	X =  -173.041  mm,	Y =   306.461  mm,	Z =     0.000  mm,
	W =  -167.372 deg,	P =    -0.003 deg,	R =  -135.227 deg
};
P[1118]{
   GP1:
	UF : 7, UT : 3,	CONFIG : 'F U T, 0, 0, 0',
	X =  -173.041  mm,	Y =   306.461  mm,	Z =     0.000  mm,
	W =  -167.372 deg,	P =    -0.003 deg,	R =  -135.227 deg
};
P[1119]{
   GP1:
	UF : 7, UT : 3,	CONFIG : 'F U T, 0, 0, 0',
	X =  -190.720  mm,	Y =   295.790  mm,	Z =     0.003  mm,
	W =  -167.372 deg,	P =    -0.002 deg,	R =  -132.163 deg
};
P[1120]{
   GP1:
	UF : 7, UT : 3,	CONFIG : 'F U T, 0, 0, 0',
	X =  -206.490  mm,	Y =   284.994  mm,	Z =     0.009  mm,
	W =  -167.373 deg,	P =    -0.002 deg,	R =  -128.960 deg
};
P[1121]{
   GP1:
	UF : 7, UT : 3,	CONFIG : 'F U T, 0, 0, 0',
	X =  -222.160  mm,	Y =   272.963  mm,	Z =     0.016  mm,
	W =  -167.373 deg,	P =    -0.001 deg,	R =  -125.844 deg
};
P[1122]{
   GP1:
	UF : 7, UT : 3,	CONFIG : 'F U T, 0, 0, 0',
	X =  -236.698  mm,	Y =   260.451  mm,	Z =     0.021  mm,
	W =  -167.374 deg,	P =     0.000 deg,	R =  -122.644 deg
};
P[1123]{
   GP1:
	UF : 7, UT : 3,	CONFIG : 'F U T, 0, 0, 0',
	X =  -249.147  mm,	Y =   248.563  mm,	Z =     0.016  mm,
	W =  -167.414 deg,	P =     0.050 deg,	R =  -119.969 deg
};
P[1124]{
   GP1:
	UF : 7, UT : 3,	CONFIG : 'F U T, 0, 0, 0',
	X =  -260.264  mm,	Y =   236.898  mm,	Z =     0.000  mm,
	W =  -167.447 deg,	P =     0.100 deg,	R =  -117.131 deg
};
P[1125]{
   GP1:
	UF : 7, UT : 3,	CONFIG : 'F U T, 0, 0, 0',
	X =  -260.264  mm,	Y =   236.898  mm,	Z =     0.000  mm,
	W =  -167.447 deg,	P =     0.100 deg,	R =  -117.131 deg
};
P[1126]{
   GP1:
	UF : 7, UT : 3,	CONFIG : 'F U T, 0, 0, 0',
	X =  -260.264  mm,	Y =   236.898  mm,	Z =     0.000  mm,
	W =  -167.447 deg,	P =     0.100 deg,	R =  -117.131 deg
};
P[1127]{
   GP1:
	UF : 7, UT : 3,	CONFIG : 'F U T, 0, 0, 0',
	X =  -260.264  mm,	Y =   236.898  mm,	Z =     0.000  mm,
	W =  -167.447 deg,	P =     0.100 deg,	R =  -117.131 deg
};
P[1128]{
   GP1:
	UF : 7, UT : 3,	CONFIG : 'F U T, 0, 0, 0',
	X =  -288.873  mm,	Y =   201.022  mm,	Z =     0.000  mm,
	W =  -167.893 deg,	P =    -0.197 deg,	R =  -110.313 deg
};
P[1129]{
   GP1:
	UF : 7, UT : 3,	CONFIG : 'F U T, 0, 0, 0',
	X =  -288.873  mm,	Y =   201.022  mm,	Z =     0.000  mm,
	W =  -167.893 deg,	P =    -0.197 deg,	R =  -110.313 deg
};
P[1130]{
   GP1:
	UF : 7, UT : 3,	CONFIG : 'F U T, 0, 0, 0',
	X =  -288.873  mm,	Y =   201.022  mm,	Z =     0.000  mm,
	W =  -167.893 deg,	P =    -0.197 deg,	R =  -110.313 deg
};
P[1131]{
   GP1:
	UF : 7, UT : 3,	CONFIG : 'F U T, 0, 0, 0',
	X =  -288.873  mm,	Y =   201.022  mm,	Z =     0.000  mm,
	W =  -167.893 deg,	P =    -0.197 deg,	R =  -110.313 deg
};
P[1132]{
   GP1:
	UF : 7, UT : 3,	CONFIG : 'F U T, 0, 0, 0',
	X =  -297.890  mm,	Y =   187.407  mm,	Z =     0.208  mm,
	W =  -168.125 deg,	P =    -1.096 deg,	R =  -107.109 deg
};
P[1133]{
   GP1:
	UF : 7, UT : 3,	CONFIG : 'F U T, 0, 0, 0',
	X =  -301.777  mm,	Y =   181.079  mm,	Z =     0.410  mm,
	W =  -168.208 deg,	P =    -1.678 deg,	R =  -106.017 deg
};
P[1134]{
   GP1:
	UF : 7, UT : 3,	CONFIG : 'F U T, 0, 0, 0',
	X =  -306.225  mm,	Y =   173.464  mm,	Z =     0.720  mm,
	W =  -168.359 deg,	P =    -1.852 deg,	R =  -104.630 deg
};
P[1135]{
   GP1:
	UF : 7, UT : 3,	CONFIG : 'F U T, 0, 0, 0',
	X =  -310.479  mm,	Y =   165.757  mm,	Z =     1.000  mm,
	W =  -168.472 deg,	P =    -1.237 deg,	R =  -103.508 deg
};
P[1136]{
   GP1:
	UF : 7, UT : 3,	CONFIG : 'F U T, 0, 0, 0',
	X =  -310.479  mm,	Y =   165.757  mm,	Z =     1.000  mm,
	W =  -168.472 deg,	P =    -1.237 deg,	R =  -103.508 deg
};
P[1137]{
   GP1:
	UF : 7, UT : 3,	CONFIG : 'F U T, 0, 0, 0',
	X =  -310.479  mm,	Y =   165.757  mm,	Z =     1.000  mm,
	W =  -168.472 deg,	P =    -1.237 deg,	R =  -103.508 deg
};
P[1138]{
   GP1:
	UF : 7, UT : 3,	CONFIG : 'F U T, 0, 0, 0',
	X =  -310.479  mm,	Y =   165.757  mm,	Z =     1.000  mm,
	W =  -168.472 deg,	P =    -1.237 deg,	R =  -103.508 deg
};
P[1139]{
   GP1:
	UF : 7, UT : 3,	CONFIG : 'F U T, 0, 0, 0',
	X =  -323.165  mm,	Y =   139.394  mm,	Z =     1.000  mm,
	W =  -167.595 deg,	P =     1.008 deg,	R =   -98.966 deg
};
P[1140]{
   GP1:
	UF : 7, UT : 3,	CONFIG : 'F U T, 0, 0, 0',
	X =  -323.165  mm,	Y =   139.394  mm,	Z =     1.000  mm,
	W =  -167.595 deg,	P =     1.008 deg,	R =   -98.966 deg
};
P[1141]{
   GP1:
	UF : 7, UT : 3,	CONFIG : 'F U T, 0, 0, 0',
	X =  -323.165  mm,	Y =   139.394  mm,	Z =     1.000  mm,
	W =  -167.595 deg,	P =     1.008 deg,	R =   -98.966 deg
};
P[1142]{
   GP1:
	UF : 7, UT : 3,	CONFIG : 'F U T, 0, 0, 0',
	X =  -323.165  mm,	Y =   139.394  mm,	Z =     1.000  mm,
	W =  -167.595 deg,	P =     1.008 deg,	R =   -98.966 deg
};
P[1143]{
   GP1:
	UF : 7, UT : 3,	CONFIG : 'F U T, 0, 0, 0',
	X =  -328.405  mm,	Y =   126.540  mm,	Z =     0.631  mm,
	W =  -167.514 deg,	P =     2.212 deg,	R =   -95.957 deg
};
P[1144]{
   GP1:
	UF : 7, UT : 3,	CONFIG : 'F U T, 0, 0, 0',
	X =  -330.738  mm,	Y =   120.311  mm,	Z =     0.385  mm,
	W =  -167.607 deg,	P =     2.141 deg,	R =   -94.815 deg
};
P[1145]{
   GP1:
	UF : 7, UT : 3,	CONFIG : 'F U T, 0, 0, 0',
	X =  -335.864  mm,	Y =   105.155  mm,	Z =     0.029  mm,
	W =  -167.677 deg,	P =     0.615 deg,	R =   -92.305 deg
};
P[1146]{
   GP1:
	UF : 7, UT : 3,	CONFIG : 'F U T, 0, 0, 0',
	X =  -337.294  mm,	Y =   100.499  mm,	Z =     0.000  mm,
	W =  -167.622 deg,	P =     0.306 deg,	R =   -92.059 deg
};
P[1147]{
   GP1:
	UF : 7, UT : 3,	CONFIG : 'F U T, 0, 0, 0',
	X =  -337.294  mm,	Y =   100.499  mm,	Z =     0.000  mm,
	W =  -167.622 deg,	P =     0.306 deg,	R =   -92.059 deg
};
P[1148]{
   GP1:
	UF : 7, UT : 3,	CONFIG : 'F U T, 0, 0, 0',
	X =  -337.294  mm,	Y =   100.499  mm,	Z =     0.000  mm,
	W =  -167.622 deg,	P =     0.306 deg,	R =   -92.059 deg
};
P[1149]{
   GP1:
	UF : 7, UT : 3,	CONFIG : 'F U T, 0, 0, 0',
	X =  -337.294  mm,	Y =   100.499  mm,	Z =     0.000  mm,
	W =  -167.622 deg,	P =     0.306 deg,	R =   -92.059 deg
};
P[1150]{
   GP1:
	UF : 7, UT : 3,	CONFIG : 'F U T, 0, 1, 0',
	X =  -347.491  mm,	Y =    55.790  mm,	Z =     0.000  mm,
	W =  -167.390 deg,	P =    -0.010 deg,	R =   -84.124 deg
};
P[1151]{
   GP1:
	UF : 7, UT : 3,	CONFIG : 'F U T, 0, 1, 0',
	X =  -347.491  mm,	Y =    55.790  mm,	Z =     0.000  mm,
	W =  -167.390 deg,	P =    -0.010 deg,	R =   -84.124 deg
};
P[1152]{
   GP1:
	UF : 7, UT : 3,	CONFIG : 'F U T, 0, 1, 0',
	X =  -347.491  mm,	Y =    55.790  mm,	Z =     0.000  mm,
	W =  -167.390 deg,	P =    -0.010 deg,	R =   -84.124 deg
};
P[1153]{
   GP1:
	UF : 7, UT : 3,	CONFIG : 'F U T, 0, 1, 0',
	X =  -347.491  mm,	Y =    55.790  mm,	Z =     0.000  mm,
	W =  -167.390 deg,	P =    -0.010 deg,	R =   -84.124 deg
};
P[1154]{
   GP1:
	UF : 7, UT : 3,	CONFIG : 'F U T, 0, 1, 0',
	X =  -349.820  mm,	Y =    38.586  mm,	Z =     0.003  mm,
	W =  -167.382 deg,	P =    -0.003 deg,	R =   -81.231 deg
};
P[1155]{
   GP1:
	UF : 7, UT : 3,	CONFIG : 'F U T, 0, 1, 0',
	X =  -351.303  mm,	Y =    21.167  mm,	Z =     0.003  mm,
	W =  -167.373 deg,	P =     0.003 deg,	R =   -78.345 deg
};
P[1156]{
   GP1:
	UF : 7, UT : 3,	CONFIG : 'F U T, 0, 1, 0',
	X =  -351.955  mm,	Y =     0.000  mm,	Z =     0.000  mm,
	W =  -167.361 deg,	P =     0.009 deg,	R =   -75.581 deg
};
P[1157]{
   GP1:
	UF : 7, UT : 3,	CONFIG : 'F U T, 0, 1, 0',
	X =  -351.955  mm,	Y =     0.000  mm,	Z =     0.000  mm,
	W =  -167.361 deg,	P =     0.009 deg,	R =   -75.581 deg
};
P[1158]{
   GP1:
	UF : 7, UT : 3,	CONFIG : 'F U T, 0, 1, 0',
	X =  -351.955  mm,	Y =     0.000  mm,	Z =     0.000  mm,
	W =  -167.361 deg,	P =     0.009 deg,	R =   -75.581 deg
};
P[1159]{
   GP1:
	UF : 7, UT : 3,	CONFIG : 'F U T, 0, 1, 0',
	X =  -351.955  mm,	Y =     0.000  mm,	Z =     0.000  mm,
	W =  -167.361 deg,	P =     0.009 deg,	R =   -75.581 deg
};
P[1160]{
   GP1:
	UF : 7, UT : 3,	CONFIG : 'F U T, 0, 1, 0',
	X =  -348.821  mm,	Y =     0.000  mm,	Z =     0.000  mm,
	W =  -167.361 deg,	P =     0.009 deg,	R =   -75.580 deg
};
P[1161]{
   GP1:
	UF : 7, UT : 3,	CONFIG : 'F U T, 0, 1, 0',
	X =  -348.821  mm,	Y =     0.000  mm,	Z =     0.000  mm,
	W =  -167.361 deg,	P =     0.009 deg,	R =   -75.580 deg
};
P[1162]{
   GP1:
	UF : 7, UT : 3,	CONFIG : 'F U T, 0, 1, 0',
	X =  -348.821  mm,	Y =     0.000  mm,	Z =     0.000  mm,
	W =  -167.361 deg,	P =     0.009 deg,	R =   -75.580 deg
};
P[1163]{
   GP1:
	UF : 7, UT : 3,	CONFIG : 'F U T, 0, 1, 0',
	X =  -348.821  mm,	Y =     0.000  mm,	Z =     0.000  mm,
	W =  -167.361 deg,	P =     0.009 deg,	R =   -75.580 deg
};
P[1164]{
   GP1:
	UF : 7, UT : 3,	CONFIG : 'F U T, 0, 1, 0',
	X =  -347.719  mm,	Y =    27.446  mm,	Z =     0.003  mm,
	W =  -167.374 deg,	P =    -0.001 deg,	R =   -79.422 deg
};
P[1165]{
   GP1:
	UF : 7, UT : 3,	CONFIG : 'F U T, 0, 1, 0',
	X =  -344.991  mm,	Y =    51.425  mm,	Z =     0.000  mm,
	W =  -167.384 deg,	P =    -0.011 deg,	R =   -83.308 deg
};
P[1166]{
   GP1:
	UF : 7, UT : 3,	CONFIG : 'F U T, 0, 1, 0',
	X =  -344.991  mm,	Y =    51.425  mm,	Z =     0.000  mm,
	W =  -167.384 deg,	P =    -0.011 deg,	R =   -83.308 deg
};
P[1167]{
   GP1:
	UF : 7, UT : 3,	CONFIG : 'F U T, 0, 1, 0',
	X =  -344.991  mm,	Y =    51.425  mm,	Z =     0.000  mm,
	W =  -167.384 deg,	P =    -0.011 deg,	R =   -83.308 deg
};
P[1168]{
   GP1:
	UF : 7, UT : 3,	CONFIG : 'F U T, 0, 1, 0',
	X =  -344.991  mm,	Y =    51.425  mm,	Z =     0.000  mm,
	W =  -167.384 deg,	P =    -0.011 deg,	R =   -83.308 deg
};
P[1169]{
   GP1:
	UF : 7, UT : 3,	CONFIG : 'F U T, 0, 0, 0',
	X =  -333.135  mm,	Y =   103.355  mm,	Z =     0.000  mm,
	W =  -167.638 deg,	P =     0.437 deg,	R =   -91.561 deg
};
P[1170]{
   GP1:
	UF : 7, UT : 3,	CONFIG : 'F U T, 0, 0, 0',
	X =  -333.135  mm,	Y =   103.355  mm,	Z =     0.000  mm,
	W =  -167.638 deg,	P =     0.437 deg,	R =   -91.561 deg
};
P[1171]{
   GP1:
	UF : 7, UT : 3,	CONFIG : 'F U T, 0, 0, 0',
	X =  -333.135  mm,	Y =   103.355  mm,	Z =     0.000  mm,
	W =  -167.638 deg,	P =     0.437 deg,	R =   -91.561 deg
};
P[1172]{
   GP1:
	UF : 7, UT : 3,	CONFIG : 'F U T, 0, 0, 0',
	X =  -333.135  mm,	Y =   103.355  mm,	Z =     0.000  mm,
	W =  -167.638 deg,	P =     0.437 deg,	R =   -91.561 deg
};
P[1173]{
   GP1:
	UF : 7, UT : 3,	CONFIG : 'F U T, 0, 0, 0',
	X =  -328.255  mm,	Y =   117.948  mm,	Z =     0.291  mm,
	W =  -167.684 deg,	P =     2.047 deg,	R =   -94.688 deg
};
P[1174]{
   GP1:
	UF : 7, UT : 3,	CONFIG : 'F U T, 0, 0, 0',
	X =  -325.878  mm,	Y =   124.367  mm,	Z =     0.545  mm,
	W =  -167.629 deg,	P =     2.346 deg,	R =   -95.800 deg
};
P[1175]{
   GP1:
	UF : 7, UT : 3,	CONFIG : 'F U T, 0, 0, 0',
	X =  -324.799  mm,	Y =   127.193  mm,	Z =     0.659  mm,
	W =  -167.621 deg,	P =     2.234 deg,	R =   -96.230 deg
};
P[1176]{
   GP1:
	UF : 7, UT : 3,	CONFIG : 'F U T, 0, 0, 0',
	X =  -319.450  mm,	Y =   140.081  mm,	Z =     1.000  mm,
	W =  -167.790 deg,	P =     0.910 deg,	R =   -98.471 deg
};
P[1177]{
   GP1:
	UF : 7, UT : 3,	CONFIG : 'F U T, 0, 0, 0',
	X =  -319.450  mm,	Y =   140.081  mm,	Z =     1.000  mm,
	W =  -167.790 deg,	P =     0.910 deg,	R =   -98.471 deg
};
P[1178]{
   GP1:
	UF : 7, UT : 3,	CONFIG : 'F U T, 0, 0, 0',
	X =  -319.450  mm,	Y =   140.081  mm,	Z =     1.000  mm,
	W =  -167.790 deg,	P =     0.910 deg,	R =   -98.471 deg
};
P[1179]{
   GP1:
	UF : 7, UT : 3,	CONFIG : 'F U T, 0, 0, 0',
	X =  -319.450  mm,	Y =   140.081  mm,	Z =     1.000  mm,
	W =  -167.790 deg,	P =     0.910 deg,	R =   -98.471 deg
};
P[1180]{
   GP1:
	UF : 7, UT : 3,	CONFIG : 'F U T, 0, 0, 0',
	X =  -308.698  mm,	Y =   162.429  mm,	Z =     1.000  mm,
	W =  -168.619 deg,	P =    -0.871 deg,	R =  -102.937 deg
};
P[1181]{
   GP1:
	UF : 7, UT : 3,	CONFIG : 'F U T, 0, 0, 0',
	X =  -308.698  mm,	Y =   162.429  mm,	Z =     1.000  mm,
	W =  -168.619 deg,	P =    -0.871 deg,	R =  -102.937 deg
};
P[1182]{
   GP1:
	UF : 7, UT : 3,	CONFIG : 'F U T, 0, 0, 0',
	X =  -308.698  mm,	Y =   162.429  mm,	Z =     1.000  mm,
	W =  -168.619 deg,	P =    -0.871 deg,	R =  -102.937 deg
};
P[1183]{
   GP1:
	UF : 7, UT : 3,	CONFIG : 'F U T, 0, 0, 0',
	X =  -308.698  mm,	Y =   162.429  mm,	Z =     1.000  mm,
	W =  -168.619 deg,	P =    -0.871 deg,	R =  -102.937 deg
};
P[1184]{
   GP1:
	UF : 7, UT : 3,	CONFIG : 'F U T, 0, 0, 0',
	X =  -304.278  mm,	Y =   170.562  mm,	Z =     0.741  mm,
	W =  -168.545 deg,	P =    -1.673 deg,	R =  -104.288 deg
};
P[1185]{
   GP1:
	UF : 7, UT : 3,	CONFIG : 'F U T, 0, 0, 0',
	X =  -299.991  mm,	Y =   177.979  mm,	Z =     0.443  mm,
	W =  -168.362 deg,	P =    -1.726 deg,	R =  -105.695 deg
};
P[1186]{
   GP1:
	UF : 7, UT : 3,	CONFIG : 'F U T, 0, 0, 0',
	X =  -288.517  mm,	Y =   196.042  mm,	Z =     0.000  mm,
	W =  -167.992 deg,	P =    -0.314 deg,	R =  -108.539 deg
};
P[1187]{
   GP1:
	UF : 7, UT : 3,	CONFIG : 'F U T, 0, 0, 0',
	X =  -288.517  mm,	Y =   196.042  mm,	Z =     0.000  mm,
	W =  -167.992 deg,	P =    -0.314 deg,	R =  -108.539 deg
};
P[1188]{
   GP1:
	UF : 7, UT : 3,	CONFIG : 'F U T, 0, 0, 0',
	X =  -288.517  mm,	Y =   196.042  mm,	Z =     0.000  mm,
	W =  -167.992 deg,	P =    -0.314 deg,	R =  -108.539 deg
};
P[1189]{
   GP1:
	UF : 7, UT : 3,	CONFIG : 'F U T, 0, 0, 0',
	X =  -288.517  mm,	Y =   196.042  mm,	Z =     0.000  mm,
	W =  -167.992 deg,	P =    -0.314 deg,	R =  -108.539 deg
};
P[1190]{
   GP1:
	UF : 7, UT : 3,	CONFIG : 'F U T, 0, 0, 0',
	X =  -255.318  mm,	Y =   237.661  mm,	Z =     0.000  mm,
	W =  -167.431 deg,	P =     0.104 deg,	R =  -118.108 deg
};
P[1191]{
   GP1:
	UF : 7, UT : 3,	CONFIG : 'F U T, 0, 0, 0',
	X =  -255.318  mm,	Y =   237.661  mm,	Z =     0.000  mm,
	W =  -167.431 deg,	P =     0.104 deg,	R =  -118.108 deg
};
P[1192]{
   GP1:
	UF : 7, UT : 3,	CONFIG : 'F U T, 0, 0, 0',
	X =  -255.318  mm,	Y =   237.661  mm,	Z =     0.000  mm,
	W =  -167.431 deg,	P =     0.104 deg,	R =  -118.108 deg
};
P[1193]{
   GP1:
	UF : 7, UT : 3,	CONFIG : 'F U T, 0, 0, 0',
	X =  -255.318  mm,	Y =   237.661  mm,	Z =     0.000  mm,
	W =  -167.431 deg,	P =     0.104 deg,	R =  -118.108 deg
};
P[1194]{
   GP1:
	UF : 7, UT : 3,	CONFIG : 'F U T, 0, 0, 0',
	X =  -244.166  mm,	Y =   249.102  mm,	Z =     0.017  mm,
	W =  -167.403 deg,	P =     0.049 deg,	R =  -120.505 deg
};
P[1195]{
   GP1:
	UF : 7, UT : 3,	CONFIG : 'F U T, 0, 0, 0',
	X =  -232.964  mm,	Y =   259.606  mm,	Z =     0.020  mm,
	W =  -167.373 deg,	P =    -0.001 deg,	R =  -123.022 deg
};
P[1196]{
   GP1:
	UF : 7, UT : 3,	CONFIG : 'F U T, 0, 0, 0',
	X =  -219.177  mm,	Y =   271.343  mm,	Z =     0.016  mm,
	W =  -167.373 deg,	P =    -0.002 deg,	R =  -126.041 deg
};
P[1197]{
   GP1:
	UF : 7, UT : 3,	CONFIG : 'F U T, 0, 0, 0',
	X =  -204.531  mm,	Y =   282.545  mm,	Z =     0.009  mm,
	W =  -167.373 deg,	P =    -0.003 deg,	R =  -129.005 deg
};
P[1198]{
   GP1:
	UF : 7, UT : 3,	CONFIG : 'F U T, 0, 0, 0',
	X =  -189.632  mm,	Y =   292.762  mm,	Z =     0.003  mm,
	W =  -167.373 deg,	P =    -0.004 deg,	R =  -132.024 deg
};
P[1199]{
   GP1:
	UF : 7, UT : 3,	CONFIG : 'F U T, 0, 0, 0',
	X =  -174.892  mm,	Y =   301.790  mm,	Z =     0.000  mm,
	W =  -167.372 deg,	P =    -0.005 deg,	R =  -135.243 deg
};
P[1200]{
   GP1:
	UF : 7, UT : 3,	CONFIG : 'F U T, 0, 0, 0',
	X =  -174.892  mm,	Y =   301.790  mm,	Z =     0.000  mm,
	W =  -167.372 deg,	P =    -0.005 deg,	R =  -135.243 deg
};
P[1201]{
   GP1:
	UF : 7, UT : 3,	CONFIG : 'F U T, 0, 0, 0',
	X =  -174.892  mm,	Y =   301.790  mm,	Z =     0.000  mm,
	W =  -167.372 deg,	P =    -0.005 deg,	R =  -135.243 deg
};
P[1202]{
   GP1:
	UF : 7, UT : 3,	CONFIG : 'F U T, 0, 0, 0',
	X =  -174.892  mm,	Y =   301.790  mm,	Z =     0.000  mm,
	W =  -167.372 deg,	P =    -0.005 deg,	R =  -135.243 deg
};
P[1203]{
   GP1:
	UF : 7, UT : 3,	CONFIG : 'F U T, 0, 0, 0',
	X =  -126.912  mm,	Y =   324.901  mm,	Z =     0.000  mm,
	W =  -167.365 deg,	P =     0.002 deg,	R =  -144.020 deg
};
P[1204]{
   GP1:
	UF : 7, UT : 3,	CONFIG : 'F U T, 0, 0, 0',
	X =  -126.912  mm,	Y =   324.901  mm,	Z =     0.000  mm,
	W =  -167.365 deg,	P =     0.002 deg,	R =  -144.020 deg
};
P[1205]{
   GP1:
	UF : 7, UT : 3,	CONFIG : 'F U T, 0, 0, 0',
	X =  -126.912  mm,	Y =   324.901  mm,	Z =     0.000  mm,
	W =  -167.365 deg,	P =     0.002 deg,	R =  -144.020 deg
};
P[1206]{
   GP1:
	UF : 7, UT : 3,	CONFIG : 'F U T, 0, 0, 0',
	X =  -126.912  mm,	Y =   324.901  mm,	Z =     0.000  mm,
	W =  -167.365 deg,	P =     0.002 deg,	R =  -144.020 deg
};
P[1207]{
   GP1:
	UF : 7, UT : 3,	CONFIG : 'F U T, 0, 0, 0',
	X =  -106.083  mm,	Y =   332.287  mm,	Z =     0.000  mm,
	W =  -167.364 deg,	P =     0.001 deg,	R =  -147.250 deg
};
P[1208]{
   GP1:
	UF : 7, UT : 3,	CONFIG : 'F U T, 0, 0, 0',
	X =   -88.319  mm,	Y =   337.433  mm,	Z =     0.000  mm,
	W =  -167.363 deg,	P =     0.000 deg,	R =  -150.913 deg
};
P[1209]{
   GP1:
	UF : 7, UT : 3,	CONFIG : 'F U T, 0, 0, 0',
	X =   -88.319  mm,	Y =   337.433  mm,	Z =     0.000  mm,
	W =  -167.363 deg,	P =     0.000 deg,	R =  -150.913 deg
};
P[1210]{
   GP1:
	UF : 7, UT : 3,	CONFIG : 'F U T, 0, 0, 0',
	X =   -88.319  mm,	Y =   337.433  mm,	Z =     0.000  mm,
	W =  -167.363 deg,	P =     0.000 deg,	R =  -150.913 deg
};
P[1211]{
   GP1:
	UF : 7, UT : 3,	CONFIG : 'F U T, 0, 0, 0',
	X =   -88.319  mm,	Y =   337.433  mm,	Z =     0.000  mm,
	W =  -167.363 deg,	P =     0.000 deg,	R =  -150.913 deg
};
P[1212]{
   GP1:
	UF : 7, UT : 3,	CONFIG : 'F U T, 0, 0, 0',
	X =   -66.816  mm,	Y =   342.344  mm,	Z =     0.000  mm,
	W =  -167.363 deg,	P =     0.000 deg,	R =  -154.099 deg
};
P[1213]{
   GP1:
	UF : 7, UT : 3,	CONFIG : 'F U T, 0, 0, 0',
	X =   -66.816  mm,	Y =   342.344  mm,	Z =     0.000  mm,
	W =  -167.363 deg,	P =     0.000 deg,	R =  -154.099 deg
};
P[1214]{
   GP1:
	UF : 7, UT : 3,	CONFIG : 'F U T, 0, 0, 0',
	X =   -66.816  mm,	Y =   342.344  mm,	Z =     0.000  mm,
	W =  -167.363 deg,	P =     0.000 deg,	R =  -154.099 deg
};
P[1215]{
   GP1:
	UF : 7, UT : 3,	CONFIG : 'F U T, 0, 0, 0',
	X =   -66.816  mm,	Y =   342.344  mm,	Z =     0.000  mm,
	W =  -167.363 deg,	P =     0.000 deg,	R =  -154.099 deg
};
P[1216]{
   GP1:
	UF : 7, UT : 3,	CONFIG : 'F U T, 0, 0, 0',
	X =   -46.005  mm,	Y =   345.765  mm,	Z =     0.000  mm,
	W =  -167.363 deg,	P =     0.000 deg,	R =  -157.374 deg
};
P[1217]{
   GP1:
	UF : 7, UT : 3,	CONFIG : 'F U T, 0, 0, 0',
	X =   -26.635  mm,	Y =   347.781  mm,	Z =     0.000  mm,
	W =  -167.364 deg,	P =     0.000 deg,	R =  -160.858 deg
};
P[1218]{
   GP1:
	UF : 7, UT : 3,	CONFIG : 'F U T, 0, 0, 0',
	X =   -26.635  mm,	Y =   347.781  mm,	Z =     0.000  mm,
	W =  -167.364 deg,	P =     0.000 deg,	R =  -160.858 deg
};
P[1219]{
   GP1:
	UF : 7, UT : 3,	CONFIG : 'F U T, 0, 0, 0',
	X =   -26.635  mm,	Y =   347.781  mm,	Z =     0.000  mm,
	W =  -167.364 deg,	P =     0.000 deg,	R =  -160.858 deg
};
P[1220]{
   GP1:
	UF : 7, UT : 3,	CONFIG : 'F U T, 0, 0, 0',
	X =   -26.635  mm,	Y =   347.781  mm,	Z =     0.000  mm,
	W =  -167.364 deg,	P =     0.000 deg,	R =  -160.858 deg
};
P[1221]{
   GP1:
	UF : 7, UT : 3,	CONFIG : 'F U T, 0, 0, 0',
	X =    26.635  mm,	Y =   347.781  mm,	Z =     0.000  mm,
	W =  -167.363 deg,	P =     0.000 deg,	R =  -169.046 deg
};
P[1222]{
   GP1:
	UF : 7, UT : 3,	CONFIG : 'F U T, 0, 0, 0',
	X =    26.635  mm,	Y =   347.781  mm,	Z =     0.000  mm,
	W =  -167.363 deg,	P =     0.000 deg,	R =  -169.046 deg
};
P[1223]{
   GP1:
	UF : 7, UT : 3,	CONFIG : 'F U T, 0, 0, 0',
	X =    26.635  mm,	Y =   347.781  mm,	Z =     0.000  mm,
	W =  -167.363 deg,	P =     0.000 deg,	R =  -169.046 deg
};
P[1224]{
   GP1:
	UF : 7, UT : 3,	CONFIG : 'F U T, 0, 0, 0',
	X =    26.635  mm,	Y =   347.781  mm,	Z =     0.000  mm,
	W =  -167.363 deg,	P =     0.000 deg,	R =  -169.046 deg
};
P[1225]{
   GP1:
	UF : 7, UT : 3,	CONFIG : 'F U T, 0, 0, 0',
	X =    45.934  mm,	Y =   345.776  mm,	Z =     0.000  mm,
	W =  -167.363 deg,	P =     0.000 deg,	R =  -172.500 deg
};
P[1226]{
   GP1:
	UF : 7, UT : 3,	CONFIG : 'F U T, 0, 0, 0',
	X =    66.816  mm,	Y =   342.344  mm,	Z =     0.000  mm,
	W =  -167.363 deg,	P =     0.000 deg,	R =  -175.771 deg
};
P[1227]{
   GP1:
	UF : 7, UT : 3,	CONFIG : 'F U T, 0, 0, 0',
	X =    66.816  mm,	Y =   342.344  mm,	Z =     0.000  mm,
	W =  -167.363 deg,	P =     0.000 deg,	R =  -175.771 deg
};
P[1228]{
   GP1:
	UF : 7, UT : 3,	CONFIG : 'F U T, 0, 0, 0',
	X =    66.816  mm,	Y =   342.344  mm,	Z =     0.000  mm,
	W =  -167.363 deg,	P =     0.000 deg,	R =  -175.771 deg
};
P[1229]{
   GP1:
	UF : 7, UT : 3,	CONFIG : 'F U T, 0, 0, 0',
	X =    66.816  mm,	Y =   342.344  mm,	Z =     0.000  mm,
	W =  -167.363 deg,	P =     0.000 deg,	R =  -175.771 deg
};
P[1230]{
   GP1:
	UF : 7, UT : 3,	CONFIG : 'F U T, 0, 0, 0',
	X =    88.319  mm,	Y =   337.433  mm,	Z =     0.000  mm,
	W =  -167.363 deg,	P =     0.000 deg,	R =  -179.012 deg
};
P[1231]{
   GP1:
	UF : 7, UT : 3,	CONFIG : 'F U T, 0, 0, 0',
	X =    88.319  mm,	Y =   337.433  mm,	Z =     0.000  mm,
	W =  -167.363 deg,	P =     0.000 deg,	R =  -179.012 deg
};
P[1232]{
   GP1:
	UF : 7, UT : 3,	CONFIG : 'F U T, 0, 0, 0',
	X =    88.319  mm,	Y =   337.433  mm,	Z =     0.000  mm,
	W =  -167.363 deg,	P =     0.000 deg,	R =  -179.012 deg
};
P[1233]{
   GP1:
	UF : 7, UT : 3,	CONFIG : 'F U T, 0, 0, 0',
	X =    88.319  mm,	Y =   337.433  mm,	Z =     0.000  mm,
	W =  -167.363 deg,	P =     0.000 deg,	R =  -179.012 deg
};
P[1234]{
   GP1:
	UF : 7, UT : 3,	CONFIG : 'F U T, 0, 0, 0',
	X =   106.083  mm,	Y =   332.287  mm,	Z =     0.000  mm,
	W =  -167.364 deg,	P =     0.000 deg,	R =   177.374 deg
};
P[1235]{
   GP1:
	UF : 7, UT : 3,	CONFIG : 'F U T, 0, 0, 0',
	X =   126.912  mm,	Y =   324.901  mm,	Z =     0.000  mm,
	W =  -167.364 deg,	P =     0.000 deg,	R =   174.134 deg
};
P[1236]{
   GP1:
	UF : 7, UT : 3,	CONFIG : 'F U T, 0, 0, 0',
	X =   126.912  mm,	Y =   324.901  mm,	Z =     0.000  mm,
	W =  -167.364 deg,	P =     0.000 deg,	R =   174.134 deg
};
P[1237]{
   GP1:
	UF : 7, UT : 3,	CONFIG : 'F U T, 0, 0, 0',
	X =   126.912  mm,	Y =   324.901  mm,	Z =     0.000  mm,
	W =  -167.364 deg,	P =     0.000 deg,	R =   174.134 deg
};
P[1238]{
   GP1:
	UF : 7, UT : 3,	CONFIG : 'F U T, 0, 0, 0',
	X =   126.912  mm,	Y =   324.901  mm,	Z =     0.000  mm,
	W =  -167.364 deg,	P =     0.000 deg,	R =   174.134 deg
};
P[1239]{
   GP1:
	UF : 7, UT : 3,	CONFIG : 'F U T, 0, 0, 0',
	X =   174.892  mm,	Y =   301.790  mm,	Z =     0.000  mm,
	W =  -167.364 deg,	P =     0.001 deg,	R =   165.335 deg
};
P[1240]{
   GP1:
	UF : 7, UT : 3,	CONFIG : 'F U T, 0, 0, 0',
	X =   174.892  mm,	Y =   301.790  mm,	Z =     0.000  mm,
	W =  -167.364 deg,	P =     0.001 deg,	R =   165.335 deg
};
P[1241]{
   GP1:
	UF : 7, UT : 3,	CONFIG : 'F U T, 0, 0, 0',
	X =   174.892  mm,	Y =   301.790  mm,	Z =     0.000  mm,
	W =  -167.364 deg,	P =     0.001 deg,	R =   165.335 deg
};
P[1242]{
   GP1:
	UF : 7, UT : 3,	CONFIG : 'F U T, 0, 0, 0',
	X =   174.892  mm,	Y =   301.790  mm,	Z =     0.000  mm,
	W =  -167.364 deg,	P =     0.001 deg,	R =   165.335 deg
};
P[1243]{
   GP1:
	UF : 7, UT : 3,	CONFIG : 'F U T, 0, 0, 0',
	X =   191.564  mm,	Y =   291.498  mm,	Z =     0.000  mm,
	W =  -167.364 deg,	P =     0.000 deg,	R =   161.703 deg
};
P[1244]{
   GP1:
	UF : 7, UT : 3,	CONFIG : 'F U T, 0, 0, 0',
	X =   208.616  mm,	Y =   279.549  mm,	Z =     0.000  mm,
	W =  -167.364 deg,	P =     0.000 deg,	R =   158.339 deg
};
P[1245]{
   GP1:
	UF : 7, UT : 3,	CONFIG : 'F U T, 0, 0, 0',
	X =   224.914  mm,	Y =   266.601  mm,	Z =     0.001  mm,
	W =  -167.364 deg,	P =     0.000 deg,	R =   154.951 deg
};
P[1246]{
   GP1:
	UF : 7, UT : 3,	CONFIG : 'F U T, 0, 0, 0',
	X =   239.976  mm,	Y =   253.131  mm,	Z =     0.000  mm,
	W =  -167.365 deg,	P =     0.000 deg,	R =   151.474 deg
};
P[1247]{
   GP1:
	UF : 7, UT : 3,	CONFIG : 'F U T, 0, 0, 0',
	X =   255.318  mm,	Y =   237.661  mm,	Z =     0.000  mm,
	W =  -167.365 deg,	P =    -0.001 deg,	R =   148.214 deg
};
P[1248]{
   GP1:
	UF : 7, UT : 3,	CONFIG : 'F U T, 0, 0, 0',
	X =   255.318  mm,	Y =   237.661  mm,	Z =     0.000  mm,
	W =  -167.365 deg,	P =    -0.001 deg,	R =   148.214 deg
};
P[1249]{
   GP1:
	UF : 7, UT : 3,	CONFIG : 'F U T, 0, 0, 0',
	X =   255.318  mm,	Y =   237.661  mm,	Z =     0.000  mm,
	W =  -167.365 deg,	P =    -0.001 deg,	R =   148.214 deg
};
P[1250]{
   GP1:
	UF : 7, UT : 3,	CONFIG : 'F U T, 0, 0, 0',
	X =   255.318  mm,	Y =   237.661  mm,	Z =     0.000  mm,
	W =  -167.365 deg,	P =    -0.001 deg,	R =   148.214 deg
};
P[1251]{
   GP1:
	UF : 7, UT : 3,	CONFIG : 'F U T, 0, 0, 0',
	X =   288.517  mm,	Y =   196.042  mm,	Z =     0.000  mm,
	W =  -167.364 deg,	P =     0.001 deg,	R =   138.644 deg
};
P[1252]{
   GP1:
	UF : 7, UT : 3,	CONFIG : 'F U T, 0, 0, 0',
	X =   288.517  mm,	Y =   196.042  mm,	Z =     0.000  mm,
	W =  -167.364 deg,	P =     0.001 deg,	R =   138.644 deg
};
P[1253]{
   GP1:
	UF : 7, UT : 3,	CONFIG : 'F U T, 0, 0, 0',
	X =   288.517  mm,	Y =   196.042  mm,	Z =     0.000  mm,
	W =  -167.364 deg,	P =     0.001 deg,	R =   138.644 deg
};
P[1254]{
   GP1:
	UF : 7, UT : 3,	CONFIG : 'F U T, 0, 0, 0',
	X =   288.517  mm,	Y =   196.042  mm,	Z =     0.000  mm,
	W =  -167.364 deg,	P =     0.001 deg,	R =   138.644 deg
};
P[1255]{
   GP1:
	UF : 7, UT : 3,	CONFIG : 'F U T, 0, 0, 0',
	X =   300.602  mm,	Y =   176.942  mm,	Z =     0.000  mm,
	W =  -167.364 deg,	P =     0.000 deg,	R =   135.546 deg
};
P[1256]{
   GP1:
	UF : 7, UT : 3,	CONFIG : 'F U T, 0, 0, 0',
	X =   309.321  mm,	Y =   161.197  mm,	Z =     0.000  mm,
	W =  -167.363 deg,	P =     0.000 deg,	R =   132.101 deg
};
P[1257]{
   GP1:
	UF : 7, UT : 3,	CONFIG : 'F U T, 0, 0, 0',
	X =   309.321  mm,	Y =   161.197  mm,	Z =     0.000  mm,
	W =  -167.363 deg,	P =     0.000 deg,	R =   132.101 deg
};
P[1258]{
   GP1:
	UF : 7, UT : 3,	CONFIG : 'F U T, 0, 0, 0',
	X =   309.321  mm,	Y =   161.197  mm,	Z =     0.000  mm,
	W =  -167.363 deg,	P =     0.000 deg,	R =   132.101 deg
};
P[1259]{
   GP1:
	UF : 7, UT : 3,	CONFIG : 'F U T, 0, 0, 0',
	X =   309.321  mm,	Y =   161.197  mm,	Z =     0.000  mm,
	W =  -167.363 deg,	P =     0.000 deg,	R =   132.101 deg
};
P[1260]{
   GP1:
	UF : 7, UT : 3,	CONFIG : 'F U T, 0, 0, 0',
	X =   318.900  mm,	Y =   141.321  mm,	Z =     0.000  mm,
	W =  -167.363 deg,	P =     0.000 deg,	R =   128.500 deg
};
P[1261]{
   GP1:
	UF : 7, UT : 3,	CONFIG : 'F U T, 0, 0, 0',
	X =   318.900  mm,	Y =   141.321  mm,	Z =     0.000  mm,
	W =  -167.363 deg,	P =     0.000 deg,	R =   128.500 deg
};
P[1262]{
   GP1:
	UF : 7, UT : 3,	CONFIG : 'F U T, 0, 0, 0',
	X =   318.900  mm,	Y =   141.321  mm,	Z =     0.000  mm,
	W =  -167.363 deg,	P =     0.000 deg,	R =   128.500 deg
};
P[1263]{
   GP1:
	UF : 7, UT : 3,	CONFIG : 'F U T, 0, 0, 0',
	X =   318.900  mm,	Y =   141.321  mm,	Z =     0.000  mm,
	W =  -167.363 deg,	P =     0.000 deg,	R =   128.500 deg
};
P[1264]{
   GP1:
	UF : 7, UT : 3,	CONFIG : 'F U T, 0, 0, 0',
	X =   327.247  mm,	Y =   120.740  mm,	Z =     0.000  mm,
	W =  -167.364 deg,	P =     0.000 deg,	R =   125.297 deg
};
P[1265]{
   GP1:
	UF : 7, UT : 3,	CONFIG : 'F U T, 0, 0, 0',
	X =   333.135  mm,	Y =   103.355  mm,	Z =     0.000  mm,
	W =  -167.365 deg,	P =    -0.001 deg,	R =   121.761 deg
};
P[1266]{
   GP1:
	UF : 7, UT : 3,	CONFIG : 'F U T, 0, 0, 0',
	X =   333.135  mm,	Y =   103.355  mm,	Z =     0.000  mm,
	W =  -167.365 deg,	P =    -0.001 deg,	R =   121.761 deg
};
P[1267]{
   GP1:
	UF : 7, UT : 3,	CONFIG : 'F U T, 0, 0, 0',
	X =   333.135  mm,	Y =   103.355  mm,	Z =     0.000  mm,
	W =  -167.365 deg,	P =    -0.001 deg,	R =   121.761 deg
};
P[1268]{
   GP1:
	UF : 7, UT : 3,	CONFIG : 'F U T, 0, 0, 0',
	X =   333.135  mm,	Y =   103.355  mm,	Z =     0.000  mm,
	W =  -167.365 deg,	P =    -0.001 deg,	R =   121.761 deg
};
P[1269]{
   GP1:
	UF : 7, UT : 3,	CONFIG : 'F U T, 0, 0, 0',
	X =   344.991  mm,	Y =    51.425  mm,	Z =     0.000  mm,
	W =  -167.364 deg,	P =     0.001 deg,	R =   113.386 deg
};
P[1270]{
   GP1:
	UF : 7, UT : 3,	CONFIG : 'F U T, 0, 0, 0',
	X =   344.991  mm,	Y =    51.425  mm,	Z =     0.000  mm,
	W =  -167.364 deg,	P =     0.001 deg,	R =   113.386 deg
};
P[1271]{
   GP1:
	UF : 7, UT : 3,	CONFIG : 'F U T, 0, 0, 0',
	X =   344.991  mm,	Y =    51.425  mm,	Z =     0.000  mm,
	W =  -167.364 deg,	P =     0.001 deg,	R =   113.386 deg
};
P[1272]{
   GP1:
	UF : 7, UT : 3,	CONFIG : 'F U T, 0, 0, 0',
	X =   344.991  mm,	Y =    51.425  mm,	Z =     0.000  mm,
	W =  -167.364 deg,	P =     0.001 deg,	R =   113.386 deg
};
P[1273]{
   GP1:
	UF : 7, UT : 3,	CONFIG : 'F U T, 0, 0, 0',
	X =   347.736  mm,	Y =    27.239  mm,	Z =     0.000  mm,
	W =  -167.364 deg,	P =     0.000 deg,	R =   109.541 deg
};
P[1274]{
   GP1:
	UF : 7, UT : 3,	CONFIG : 'F U T, 0, 0, 0',
	X =   348.821  mm,	Y =     0.000  mm,	Z =     0.000  mm,
	W =  -167.364 deg,	P =    -0.001 deg,	R =   105.687 deg
};
P[1275]{
   GP1:
	UF : 7, UT : 3,	CONFIG : 'F U T, 0, 0, 0',
	X =   348.821  mm,	Y =     0.000  mm,	Z =     0.000  mm,
	W =  -167.364 deg,	P =    -0.001 deg,	R =   105.687 deg
};
P[1276]{
   GP1:
	UF : 7, UT : 3,	CONFIG : 'F U T, 0, 0, 0',
	X =   348.821  mm,	Y =     0.000  mm,	Z =     0.000  mm,
	W =  -167.364 deg,	P =    -0.001 deg,	R =   105.687 deg
};
P[1277]{
   GP1:
	UF : 7, UT : 3,	CONFIG : 'F U T, 0, 0, 0',
	X =   348.821  mm,	Y =     0.000  mm,	Z =     0.000  mm,
	W =  -167.364 deg,	P =    -0.001 deg,	R =   105.687 deg
};
P[1278]{
   GP1:
	UF : 7, UT : 3,	CONFIG : 'F U T, 0, 0, 0',
	X =   345.686  mm,	Y =     0.000  mm,	Z =     0.000  mm,
	W =  -167.364 deg,	P =    -0.001 deg,	R =   105.687 deg
};
P[1279]{
   GP1:
	UF : 7, UT : 3,	CONFIG : 'F U T, 0, 0, 0',
	X =   345.686  mm,	Y =     0.000  mm,	Z =     0.000  mm,
	W =  -167.364 deg,	P =    -0.001 deg,	R =   105.687 deg
};
P[1280]{
   GP1:
	UF : 7, UT : 3,	CONFIG : 'F U T, 0, 0, 0',
	X =   345.686  mm,	Y =     0.000  mm,	Z =     0.000  mm,
	W =  -167.364 deg,	P =    -0.001 deg,	R =   105.687 deg
};
P[1281]{
   GP1:
	UF : 7, UT : 3,	CONFIG : 'F U T, 0, 0, 0',
	X =   345.686  mm,	Y =     0.000  mm,	Z =     0.000  mm,
	W =  -167.364 deg,	P =    -0.001 deg,	R =   105.687 deg
};
P[1282]{
   GP1:
	UF : 7, UT : 3,	CONFIG : 'F U T, 0, 0, 0',
	X =   344.660  mm,	Y =    26.365  mm,	Z =     0.000  mm,
	W =  -167.364 deg,	P =     0.000 deg,	R =   109.418 deg
};
P[1283]{
   GP1:
	UF : 7, UT : 3,	CONFIG : 'F U T, 0, 0, 0',
	X =   342.332  mm,	Y =    47.913  mm,	Z =     0.000  mm,
	W =  -167.364 deg,	P =     0.001 deg,	R =   113.455 deg
};
P[1284]{
   GP1:
	UF : 7, UT : 3,	CONFIG : 'F U T, 0, 0, 0',
	X =   342.332  mm,	Y =    47.913  mm,	Z =     0.000  mm,
	W =  -167.364 deg,	P =     0.001 deg,	R =   113.455 deg
};
P[1285]{
   GP1:
	UF : 7, UT : 3,	CONFIG : 'F U T, 0, 0, 0',
	X =   342.332  mm,	Y =    47.913  mm,	Z =     0.000  mm,
	W =  -167.364 deg,	P =     0.001 deg,	R =   113.455 deg
};
P[1286]{
   GP1:
	UF : 7, UT : 3,	CONFIG : 'F U T, 0, 0, 0',
	X =   342.332  mm,	Y =    47.913  mm,	Z =     0.000  mm,
	W =  -167.364 deg,	P =     0.001 deg,	R =   113.455 deg
};
P[1287]{
   GP1:
	UF : 7, UT : 3,	CONFIG : 'F U T, 0, 0, 0',
	X =   329.241  mm,	Y =   105.355  mm,	Z =     0.000  mm,
	W =  -167.365 deg,	P =    -0.001 deg,	R =   123.426 deg
};
P[1288]{
   GP1:
	UF : 7, UT : 3,	CONFIG : 'F U T, 0, 0, 0',
	X =   329.241  mm,	Y =   105.355  mm,	Z =     0.000  mm,
	W =  -167.365 deg,	P =    -0.001 deg,	R =   123.426 deg
};
P[1289]{
   GP1:
	UF : 7, UT : 3,	CONFIG : 'F U T, 0, 0, 0',
	X =   329.241  mm,	Y =   105.355  mm,	Z =     0.000  mm,
	W =  -167.365 deg,	P =    -0.001 deg,	R =   123.426 deg
};
/END
